// TEST/TestPackage/Templates/Internal/FB_BACnet_Server_NC01
// Notification Classes (Sample 01: Beckhoff)	
FUNCTION_BLOCK FB_BACnet_Server_NC01 EXTENDS FB_BACnet_View
VAR CONSTANT
	iAlarmModeFirst		: INT		:= 1;
	iAlarmModeLast		: INT		:= 3;
END_VAR
VAR
	// Event Typ "Alarm":
	aNCAlm_LifeSafety		: ARRAY[iAlarmModeFirst .. iAlarmModeLast] OF FB_BACnet_NC := [
								(
									iParent									:= THIS^,
									nObjectInstance							:= 12,
									nNotificationClass						:= 12,
									sObjectName								:= '\/NC12',
									sDescription							:= '\/Meldeklasse - Alarm Lebensgefahr (Einfach)',
									aAckRequired							:= [ TRUE, TRUE, FALSE ],
									aPriority								:= [ 10, 11, 12 ]),
								(
									iParent									:= THIS^,
									nObjectInstance							:= 11,
									nNotificationClass						:= 11,
									sObjectName								:= '\/NC11',
									sDescription							:= '\/Meldeklasse - Alarm Lebensgefahr (Standard)',
									aAckRequired							:= [ TRUE, TRUE, FALSE ],
									aPriority								:= [ 13, 14, 15 ]),
								(
									iParent									:= THIS^,
									nObjectInstance							:= 10,
									nNotificationClass						:= 10,
									sObjectName								:= '\/NC10',
									sDescription							:= '\/Meldeklasse - Alarm Lebensgefahr (Erweitert)',
									aAckRequired							:= [ TRUE, TRUE, TRUE ],
									aPriority								:= [ 16, 17, 18 ])
							];
							
	aNCAlm_Technical		: ARRAY[iAlarmModeFirst .. iAlarmModeLast] OF FB_BACnet_NC := [
								(
									iParent									:= THIS^,
									nObjectInstance							:= 22,
									nNotificationClass						:= 22,
									sObjectName								:= '\/NC22',
									sDescription							:= '\/Meldeklasse - Technischer Alarm (Einfach)',
									aAckRequired							:= [ TRUE, TRUE, FALSE ],
									aPriority								:= [ 20, 21, 22 ]),
								(
									iParent									:= THIS^,
									nObjectInstance							:= 21,
									nNotificationClass						:= 21,
									sObjectName								:= '\/NC21',
									sDescription							:= '\/Meldeklasse - Technischer Alarm (Standard)',
									aAckRequired							:= [ TRUE, TRUE, FALSE ],
									aPriority								:= [ 23, 24, 25 ]),
								(
									iParent									:= THIS^,
									nObjectInstance							:= 20,
									nNotificationClass						:= 20,
									sObjectName								:= '\/NC20',
									sDescription							:= '\/Meldeklasse - Technischer Alarm (Erweitert)',
									aAckRequired							:= [ TRUE, TRUE, TRUE ],
									aPriority								:= [ 26, 27, 28 ])
							];
							
	// Event Typ "Disturb":
	aNCDstb				: ARRAY[iAlarmModeFirst .. iAlarmModeLast] OF FB_BACnet_NC := [
								(
									iParent									:= THIS^,
									nObjectInstance							:= 52,
									nNotificationClass						:= 52,
									sObjectName								:= '\/NC52',
									sDescription							:= '\/Meldeklasse - Störung (Einfach)',
									aAckRequired							:= [ TRUE, TRUE, FALSE ],
									aPriority								:= [ 50, 51, 52 ]),
								(
									iParent									:= THIS^,
									nObjectInstance							:= 51,
									nNotificationClass						:= 51,
									sObjectName								:= '\/NC51',
									sDescription							:= '\/Meldeklasse - Störung (Standard)',
									aAckRequired							:= [ TRUE, TRUE, FALSE ],
									aPriority								:= [ 53, 54, 55 ]),
								(
									iParent									:= THIS^,
									nObjectInstance							:= 50,
									nNotificationClass						:= 50,
									sObjectName								:= '\/NC50',
									sDescription							:= '\/Meldeklasse - Störung (Erweitert)',
									aAckRequired							:= [ TRUE, TRUE, TRUE ],
									aPriority								:= [ 56, 57, 58 ])
							];
							
	// Event Typ "Maintenance":
	aNCMntn				: ARRAY[iAlarmModeFirst .. iAlarmModeLast] OF FB_BACnet_NC := [
								(
									iParent									:= THIS^,
									nObjectInstance							:= 92,
									nNotificationClass						:= 92,
									sObjectName								:= '\/NC92',
									sDescription							:= '\/Meldeklasse - Wartung (Einfach)',
									aAckRequired							:= [ TRUE, TRUE, FALSE ],
									aPriority								:= [ 90, 91, 92 ]),
								(
									iParent									:= THIS^,
									nObjectInstance							:= 91,
									nNotificationClass						:= 91,
									sObjectName								:= '\/NC91',
									sDescription							:= '\/Meldeklasse - Wartung (Standard)',
									aAckRequired							:= [ TRUE, TRUE, FALSE ],
									aPriority								:= [ 93, 94, 95 ]),
								(
									iParent									:= THIS^,
									nObjectInstance							:= 90,
									nNotificationClass						:= 90,
									sObjectName								:= '\/NC90',
									sDescription							:= '\/Meldeklasse - Wartung (Erweitert)',
									aAckRequired							:= [ TRUE, TRUE, TRUE ],
									aPriority								:= [ 96, 97, 98 ])
							];
							
	// Event Typ "Notification":
	aNCNtfy				: ARRAY[iAlarmModeFirst .. iAlarmModeLast] OF FB_BACnet_NC := [
								(
									iParent									:= THIS^,
									nObjectInstance							:= 132,
									nNotificationClass						:= 132,
									sObjectName								:= '\/NC132',
									sDescription							:= '\/Meldeklasse - Benachrichtigung (Einfach)',
									aAckRequired							:= [ TRUE, TRUE, FALSE ],
									aPriority								:= [ 130, 131, 132 ]),
								(
									iParent									:= THIS^,
									nObjectInstance							:= 131,
									nNotificationClass						:= 131,
									sObjectName								:= '\/NC131',
									sDescription							:= '\/Meldeklasse - Benachrichtigung (Standard)',
									aAckRequired							:= [ TRUE, TRUE, FALSE ],
									aPriority								:= [ 133, 134, 135 ]),
								(
									iParent									:= THIS^,
									nObjectInstance							:= 130,
									nNotificationClass						:= 130,
									sObjectName								:= '\/NC130',
									sDescription							:= '\/Meldeklasse - Benachrichtigung (Erweitert)',
									aAckRequired							:= [ TRUE, TRUE, TRUE ],
									aPriority								:= [ 136, 137, 138 ])
							];
							
	// Event Typ "Other":	
	aNCOthr				: ARRAY[iAlarmModeFirst .. iAlarmModeLast] OF FB_BACnet_NC := [
								(
									iParent									:= THIS^,
									nObjectInstance							:= 182,
									nNotificationClass						:= 182,
									sObjectName								:= '\/NC182',
									sDescription							:= '\/Meldeklasse - Sonstiges (Einfach)',
									aAckRequired							:= [ TRUE, TRUE, FALSE ],
									aPriority								:= [ 180, 181, 182 ]),
								(
									iParent									:= THIS^,
									nObjectInstance							:= 181,
									nNotificationClass						:= 181,
									sObjectName								:= '\/NC181',
									sDescription							:= '\/Meldeklasse - Sonstiges (Standard)',
									aAckRequired							:= [ TRUE, TRUE, FALSE ],
									aPriority								:= [ 183, 184, 185 ]),
								(
									iParent									:= THIS^,
									nObjectInstance							:= 180,
									nNotificationClass						:= 180,
									sObjectName								:= '\/NC180',
									sDescription							:= '\/Meldeklasse - Sonstiges (Erweitert)',
									aAckRequired							:= [ TRUE, TRUE, TRUE ],
									aPriority								:= [ 186, 187, 188 ])
							];
END_VAR
VAR
	iValTmp						: INT;
	iTemp						: INT;
END_VAR

SUPER^();

FOR iTemp := iAlarmModeFirst TO iAlarmModeLast DO
	aNCAlm_LifeSafety[iTemp]();
	aNCAlm_Technical[iTemp]();
	aNCDstb[iTemp]();
	aNCMntn[iTemp]();
	aNCNtfy[iTemp]();
	aNCOthr[iTemp]();
END_FOR

END_FUNCTION_BLOCK

// TEST/TestPackage/TestFBs/RT/FB_ArrayHtgCir
FUNCTION_BLOCK FB_ArrayHtgCir EXTENDS FB_BACnet_View
VAR_INPUT
	iCycleCount				: UINT;
END_VAR
VAR
	iTemp					: INT;
	aPlants					: ARRAY [1..MAX_PLANT] OF FB_Bnet_H_HtgCir_01;

	iCycleMOD				: UINT := 1;
	iLoopTo					: INT := MAX_PLANT;
END_VAR
VAR CONSTANT
	//MAX_PLANT				: INT := 29;			// Entspricht 1021 Ibjekte
	MAX_PLANT				: INT := 1;
END_VAR

SUPER^();

IF ((iCycleCount MOD iCycleMOD) = 0) THEN
	FOR iTemp := 1 TO iLoopTo DO
		aPlants[iTemp]();
	END_FOR
END_IF

METHOD FB_init : BOOL
VAR_INPUT
	bInitRetains : BOOL; // if TRUE, the retain variables are initialized (warm start / cold start)
	bInCopyCode : BOOL;  // if TRUE, the instance afterwards gets moved into the copy code (online change)
END_VAR
sObjectName		:= 'Test Heizkreise';
sDescription	:= 'Array mit vielen Heizkreisen';

FOR iTemp := 1 TO MAX_PLANT DO
	aPlants[iTemp].Parent		:= THIS^;
	aPlants[iTemp].sObjectName 	:= CONCAT('HtgCir', TO_STRING(iTemp));
	aPlants[iTemp].sDescription	:= CONCAT('Heizkreis ', TO_STRING(iTemp));
END_FOR
END_METHOD

END_FUNCTION_BLOCK

// TEST/TestPackage/TestFBs/RT/FB_ArrayTest
FUNCTION_BLOCK FB_ArrayTest EXTENDS FB_BACnet_View
VAR_INPUT
	iCycleCount				: UINT;
END_VAR
VAR					
	iTemp					: INT;
	BVObjects				: ARRAY [1..MAX_OBJECT] OF FB_BACnet_BV;

	iCycleMOD				: UINT := 1;
	iLoopTo					: INT := MAX_OBJECT;
END_VAR
VAR CONSTANT
	MAX_OBJECT : INT := 1000;
END_VAR

SUPER^();

IF ((iCycleCount MOD iCycleMOD) = 0) THEN
	FOR iTemp := 1 TO iLoopTo DO
		BVObjects[iTemp]();
	END_FOR
END_IF

METHOD FB_init : BOOL
VAR_INPUT
	bInitRetains : BOOL; // if TRUE, the retain variables are initialized (warm start / cold start)
	bInCopyCode : BOOL;  // if TRUE, the instance afterwards gets moved into the copy code (online change)
END_VAR
sObjectName		:= 'TestArray';
sDescription	:= 'Array mit vielen Objekten';

FOR iTemp := 1 TO MAX_OBJECT DO
	BVObjects[iTemp].Parent						:= THIS^;
//	BVObjects[iTemp].sObjectName 				:= CONCAT('BV üäß', TO_STRING(iTemp));
//	BVObjects[iTemp].sDescription				:= CONCAT('Binary Value üäß ', TO_STRING(iTemp));
//	
//	BVObjects[iTemp].sActiveText				:= '€ ÄÄÄ üß';
//	BVObjects[iTemp].sInactiveText				:= 'Money money $$ ÄÄÄ üß';
END_FOR
END_METHOD

END_FUNCTION_BLOCK

// TEST/TestPackage/TestFBs/FB_ClientTest
FUNCTION_BLOCK FB_ClientTest
VAR_INPUT CONSTANT
	AV_1 : FB_BACnetRM_AV := (Client:=Client,nObjectInstance:=1);
	AV_2 : FB_BACnetRM_AV := (Client:=Client,nObjectInstance:=2);
	AV_3 : FB_BACnetRM_AV := (Client:=Client,nObjectInstance:=3);
	AV_4 : FB_BACnetRM_AV := (Client:=Client,nObjectInstance:=4);
	AV_5 : FB_BACnetRM_AV := (Client:=Client,nObjectInstance:=5);
	AV_6 : FB_BACnetRM_AV := (Client:=Client,nObjectInstance:=6);
	AV_7 : FB_BACnetRM_AV := (Client:=Client,nObjectInstance:=7);
	AV_8 : FB_BACnetRM_AV := (Client:=Client,nObjectInstance:=8);
	AV_9 : FB_BACnetRM_AV := (Client:=Client,nObjectInstance:=9);
	AV_10: FB_BACnetRM_AV := (Client:=Client,nObjectInstance:=10);
	AV_11: FB_BACnetRM_AV := (Client:=Client,nObjectInstance:=11);
	AV_12: FB_BACnetRM_AV := (Client:=Client,nObjectInstance:=12);
END_VAR
VAR
	Client : FB_BACnet_Client := (eReadMode:=E_BACnet_CommMode.eRp);
END_VAR

Client();
AV_1();
AV_2();
AV_3();
AV_4();
AV_5();
AV_6();
AV_7();
AV_8();
AV_9();
AV_10();
AV_11();
AV_12();

END_FUNCTION_BLOCK

// TEST/TestPackage/_MAIN
PROGRAM _MAIN
VAR
	wDummy			AT %I*	: WORD;
	
	bKillMe11				: BOOL;
END_VAR
VAR
	bInit					: BOOL := TRUE;
	nCycles					: UDINT;
END_VAR
VAR
	bManualWritePersistent	: BOOL;
	tAutoWritePersistent	: TON						:= (PT := T#20S);
	wPersistentData			: FB_WritePersistentData	:= (PORT:=TwinCAT_SystemInfoVarList._AppInfo.AdsPort, TMOUT:=T#1S, MODE:=E_PersistentMode.SPDM_2PASS);
END_VAR

nCycles := (nCycles+1);
IF (bInit) THEN
	bInit := FALSE;
END_IF

// Persistent data:
tAutoWritePersistent(IN := (NOT tAutoWritePersistent.Q));
IF (bManualWritePersistent) OR (tAutoWritePersistent.Q) THEN
	bManualWritePersistent := FALSE;
	wPersistentData(START:=TRUE);
ELSE
	wPersistentData();
	IF (NOT wPersistentData.BUSY) THEN
		wPersistentData.START:=FALSE;
	END_IF
END_IF



// Sample programs:
// Uncomment to execute samples:
//////////////////////////////////////////////////

//CLIENT();
//PLANT_DEMO();
//MAIN_PRG02();
//PERFORMANCE();
//PERFORMANCE_MIX();
RT();
//DYN_OBJECTS();

END_PROGRAM

// TEST/TestPackage/PLANT_DEMO
PROGRAM PLANT_DEMO
VAR
	fbStatHeatingCir	: FB_Bnet_H_HtgCir_01		:= (sObjectName				:= 'HTGCIR01',
														sDescription			:= '\/Statische Heizung',
														Pu := (
															sObjectName			:= '\/TEST01_PU01',
															Dst := (
																sObjectName		:= '\/DST01')));
																
	fbFlHeatingCir		: FB_Bnet_H_HtgCir_01		:= (sObjectName				:= 'HTGCIR02',
														sDescription			:= '\/Fußbodenheizung');
																
	fbRoom3				: FB_Bnet_H_HtgCir_01		:= (sObjectName				:= 'HTGCIR03',
														sDescription			:= '\/Heizung Raum 3');
END_VAR

fbStatHeatingCir();
fbFlHeatingCir();
fbRoom3();

METHOD FB_init : BOOL
VAR_INPUT
	bInitRetains : BOOL; // if TRUE, the retain variables are initialized (warm start / cold start)
	bInCopyCode : BOOL;  // if TRUE, the instance afterwards gets moved into the copy code (online change)
END_VAR
fbStatHeatingCir.Pu.sObjectName			:= '\/TEST01_PU01';
fbStatHeatingCir.Pu.sObjectName			:= '\/TEST01_PU01';
fbStatHeatingCir.Pu.sObjectName			:= '\/TEST01_PU01';
fbStatHeatingCir.Pu.sObjectName			:= '\/TEST01_PU01';
fbStatHeatingCir.Pu.sObjectName			:= '\/TEST01_PU01';
END_METHOD

END_PROGRAM

// TEST/TestPackage/PERFORMANCE
PROGRAM PERFORMANCE
// Test für RT-Objekte:
VAR
	//fbHtgCirArray : FB_ArrayHtgCir;
	fbObjArray : FB_ArrayTest;
	
	bStop : BOOL;
END_VAR


// Test für RT-Objekte:
//fbHtgCirArray();
IF NOT bStop THEN
	fbObjArray();
END_IF

END_PROGRAM

// TEST/TestPackage/RT
// Dieses Programm testet die RT-Bausteine, welche der LIB-Variante nachempfunden sind.
PROGRAM RT
VAR
	bKillMe1 : BOOL;
	_hRes : HRESULT;
	tTemp : T_MaxString;
END_VAR
VAR_INPUT
	nLibNode_UpdateCount				: UDINT;
	fbLibNode							: FB_BACnet_View := (
											eNodeType								:= E_BACnet_NodeType.eArea,
											sObjectName								:= '\/LibNde',
											sDescription							:= '\/Test RT-Lib Node');
END_VAR
// --- Analog: ---------------------------------------------------------------------------------------------------------------------------------------
VAR_INPUT
	fbANode								: FB_BACnet_View := (
											iParent									:= fbLibNode,
											eNodeType								:= E_BACnet_NodeType.eArea,
											sObjectName								:= '\/A',
											sDescription							:= '\/Analog');

	AV									: FB_BACnet_AV := (
											iParent									:= fbANode,
											nObjectInstance							:= 115,
											sObjectName								:= '\/AV 01',
											sDescription							:= '\/Analog Value Test 1 öäü',
											eUnit									:= E_BA_Unit.eOther_Percent,
											bHighLimitEnable						:= TRUE,
											fHighLimit								:= 50,
											bLowLimitEnable							:= TRUE,
											fLowLimit								:= 10,
											nNotificationClass						:= 11,
											aEventEnable							:= [ TRUE, TRUE, FALSE ],
											aEventMessageTextsConfig				:= [ '\/Ausgelöst', '\/Fehler', '\/Normal' ]);

	// Intention:						Value
	// Priorities						5P
	AV5P_TestEnSfty				AT %I*	: BOOL; // Test: Safety ist von PLC aus immer beschaltet
	AV5P								: FB_BACnet_AV_5P := (
											iParent									:= fbANode,
											sDescription							:= '\/Analog Value 5Prio',
											eUnit									:= E_BA_Unit.eOther_Percent,
											bEnPgm									:= TRUE,
											fValPgm									:= 10.0);
											
	// Intention:						Value for Display
	// Operation:						Display
	AVDsp								: FB_BACnet_AV_Disp := (
											iParent									:= fbANode,
											sDescription							:= '\/Test AV Display',
											eUnit									:= E_BA_Unit.eOther_Percent);	
	
	// Intention:						Value for Setpoint
	// Operation:						Setpoint
	AVSp								: FB_BACnet_AV_Setp := (
											iParent									:= fbANode,
											sDescription							:= '\/Test AV Setpoint',
											eUnit									:= E_BA_Unit.eTime_Hours,
											fValue									:= 168);

	AI_TSenRaw_State			AT %I*	: USINT;
	AI_TSenRaw_DataIn			AT %I*	: INT;
	AI_TSenRaw							: FB_BACnet_AI_Raw := (
											iParent									:= fbANode,
											sDescription							:= '\/Test AI Fühler (Raw)',
											sDeviceType								:= 'Fühler',
											eUnit									:= E_BA_Unit.eOther_Percent,
											fResolution								:= 0.003814755,
											fScaleOffset							:= 0.0,
											fHighLimit								:= 150,
											fLowLimit								:= -500,
											nNotificationClass						:= 10,
											aEventEnable							:= [ TRUE, TRUE, FALSE ],
											aEventMessageTextsConfig				:= [ '\/Ausgelöst', '\/Fehler', '\/Normal' ]);

	// Intention:						Input
	// Hardware:						Process
	AI_TSenProc_Value					: REAL := 50.0;
	AI_TSenProc							: FB_BACnet_AI := (
											iParent									:= fbANode,
											sDescription							:= '\/Test AI (Prozesswert)',
											eUnit									:= E_BA_Unit.eOther_Percent,
											fHighLimit								:= 150,
											fLowLimit								:= -500,
											nNotificationClass						:= 10,
											aEventEnable							:= [ TRUE, TRUE, FALSE ],
											aEventMessageTextsConfig				:= [ '\/Ausgelöst', '\/Fehler', '\/Normal' ]);

	// Intention:						Input
	// Hardware:						I/O
	AI_TSenIO_IOBusState		AT %Q*	: UINT := 0;
	AI_TSenIO							: FB_BACnet_AI_IO := (
											iParent									:= fbANode,
											sDescription							:= '\/Test AI Fühler (IO)',
											sDeviceType								:= 'Fühler',
											eUnit									:= E_BA_Unit.eOther_Percent,
											fResolution								:= 0.003814755,
											fScaleOffset							:= 0.0,
											fHighLimit								:= 150,
											fLowLimit								:= -500,
											nIoBusNr								:= 0,
											nNotificationClass						:= 10,
											aEventEnable							:= [ TRUE, TRUE, FALSE ],
											aEventMessageTextsConfig				:= [ '\/Ausgelöst', '\/Fehler', '\/Normal' ]);

	// Intention:						Input for Display
	// Operation:						Display
	// Hardware:						I/O
	// Parameter:						EventDetectionEnable = FALSE
	AIDsp_TSenIO						: FB_BACnet_AI_IO := (
											iParent									:= fbANode,
											sDescription							:= '\/Test AI Display Fühler (IO)',
											sDeviceType								:= 'Fühler',
											eUnit									:= E_BA_Unit.eOther_Percent,
											bEventDetectionEnable					:= FALSE);

	AO_Cmd_RlbtyPgm						: E_BA_Reliability;
	AO_Cmd_RawOvrrd						: BOOL;
	AO_Cmd								: FB_BACnet_AO := (
											iParent									:= fbANode,
											sDescription							:= '\/Befehl AO',
											sDeviceType								:= 'Ausgang',
											eUnit									:= E_BA_Unit.eOther_Percent,
											fResolution								:= 0.003051851,
											fScaleOffset							:= 0.0,
											fHighLimit								:= 150,
											fLowLimit								:= -50,
											nNotificationClass						:= 10,
											aEventEnable							:= [ TRUE, TRUE, FALSE ],
											aEventMessageTextsConfig				:= [ '\/Ausgelöst', '\/Fehler', '\/Normal' ]);

	AO_CmdRaw_Out				AT %Q*	: INT;
	AO_CmdRaw							: FB_BACnet_AO_Raw := (
											iParent									:= fbANode,
											sDescription							:= '\/Befehl AO (Raw)',
											sDeviceType								:= 'Ausgang',
											eUnit									:= E_BA_Unit.eOther_Percent,
											fResolution								:= 0.003051851,
											fScaleOffset							:= 0.0,
											fHighLimit								:= 150,
											fLowLimit								:= -50,
											nNotificationClass						:= 10,
											aEventEnable							:= [ TRUE, TRUE, FALSE ],
											aEventMessageTextsConfig				:= [ '\/Ausgelöst', '\/Fehler', '\/Normal' ]);

	AO_CmdIORaw							: FB_BACnet_AO_IO := (
											iParent									:= fbANode,
											sDescription							:= '\/Befehl AO (IO)',
											sDeviceType								:= 'Ausgang',
											eUnit									:= E_BA_Unit.eOther_Percent,
											fResolution								:= 0.003051851,
											fScaleOffset							:= 0.0,
											fHighLimit								:= 150,
											fLowLimit								:= -50,
											nNotificationClass						:= 10,
											aEventEnable							:= [ TRUE, TRUE, FALSE ],
											aEventMessageTextsConfig				:= [ '\/Ausgelöst', '\/Fehler', '\/Normal' ]);

	AO_Cmd5P_RlbtyPgm					: E_BA_Reliability;
	AO_Cmd5P_RawOvrrd					: BOOL;
	AO_Cmd5P							: FB_BACnet_AO_5P := (
											iParent									:= fbANode,
											sDescription							:= '\/Analog Befehl 5Prio',
											eUnit									:= E_BA_Unit.eOther_Percent);

	AO_CmdRaw5P_State			AT %I*	: USINT;
	AO_CmdRaw5P_Out				AT %Q*	: INT;
	AO_CmdRaw5P							: FB_BACnet_AO_Raw5P := (
											iParent									:= fbANode,
											sDescription							:= '\/Analog Befehl 5Prio (Raw)',
											eUnit									:= E_BA_Unit.eOther_Percent);

	// Intention:						Output
	// Hardware:						I/O
	// Priorities						5P
	AO_CmdIO5P							: FB_BACnet_AO_IO5P := (
											iParent									:= fbANode,
											sDescription							:= '\/Analog Befehl 5Prio (IO)',
											eUnit									:= E_BA_Unit.eOther_Percent);

	// Intention:						Output for Display
	// Operation:						Display
	// Hardware:						I/O
	// Parameter:						EventDetectionEnable = FALSE
	AODisp_CmdIO5P						: FB_BACnet_AO_IO5P := (
											iParent									:= fbANode,
											sDescription							:= '\/Analog Befehl 5Prio Display (IO)',
											eUnit									:= E_BA_Unit.eOther_Percent,
											bEventDetectionEnable					:= FALSE);
											
	AO_CmdIO							: FB_BACnet_AO_IO := (
											iParent									:= fbANode,
											sDescription							:= '\/Analog Befehl (IO)',
											eUnit									:= E_BA_Unit.eOther_Percent);
END_VAR
// --- Binary: ---------------------------------------------------------------------------------------------------------------------------------------
VAR_INPUT
	fbBNode								: FB_BACnet_View := (
											iParent									:= fbLibNode,
											eNodeType								:= E_BACnet_NodeType.eArea,
											sObjectName								:= '\/B',
											sDescription							:= '\/Binary');
											
	BV									: FB_BACnet_BV := (
											iParent									:= fbBNode,
											nObjectInstance							:= 99,
											sDescription							:= '\/Test BV',
											bAlarmValue								:= FALSE);

	// Intention:						Value
	// Priorities						5P
	BV5P								: FB_BACnet_BV_5P := (
											iParent									:= fbBNode,
											sDescription							:= '\/Binary Value 5Prio');
											
	// Intention:						Value for Display
	// Operation:						Display
	BVDsp								: FB_BACnet_BV_Disp := (
											iParent									:= fbBNode,
											sDescription							:= '\/Test BV Display',
											sInactiveText							:= 'Aus',
											sActiveText								:= 'Ein');
	
	// Intention:						Value for Setpoint
	// Operation:						Setpoint
	BVSp								: FB_BACnet_BV_Setp := (
											iParent									:= fbBNode,
											sDescription							:= '\/Test BV Setpoint',
											sInactiveText							:= 'Aus',
											sActiveText								:= 'Ein',
											bValue									:= TRUE);

	BI_DstbRaw_In				AT %I*	: BOOL;
	BI_DstbRaw							: FB_BACnet_BI_Raw := (
											iParent									:= fbBNode,
											sDescription							:= '\/Test BI Disturb (Raw)',
											sDeviceType								:= 'Sicherung',
											sInactiveText							:= 'Normal',
											sActiveText								:= 'Ausgelöst',
											ePolarity								:= E_BA_Polarity.eReverse,
											nNotificationClass						:= 10,
											aEventEnable							:= [ TRUE, TRUE, FALSE ],
											aEventMessageTextsConfig				:= [ '\/Ausgelöst', '\/Fehler', '\/Normal' ]);
											
	// Intention:						Input
	// Hardware:						I/O
	BI_DstbIO							: FB_BACnet_BI_IO := (
											iParent									:= fbBNode,
											sDescription							:= '\/Test BI Disturb (IO)',
											sDeviceType								:= 'Sicherung',
											sInactiveText							:= 'Normal',
											sActiveText								:= 'Ausgelöst',
											ePolarity								:= E_BA_Polarity.eReverse,
											nNotificationClass						:= 10,
											aEventEnable							:= [ TRUE, TRUE, FALSE ],
											aEventMessageTextsConfig				:= [ '\/Ausgelöst', '\/Fehler', '\/Normal' ]);

	// Intention:						Input for Display
	// Operation:						Display
	// Hardware:						I/O
	// Parameter:						EventDetectionEnable = FALSE
	BIDsp_SwiIO							: FB_BACnet_BI_IO := (
											iParent									:= fbBNode,
											sDescription							:= '\/Test BI Schalter Display (IO)',
											sDeviceType								:= 'Sicherung',
											sInactiveText							:= 'Normal',
											sActiveText								:= 'Ausgelöst',
											ePolarity								:= E_BA_Polarity.eReverse,
											bEventDetectionEnable					:= FALSE);

	BO_Cmd_RlbtyPgm						: E_BA_Reliability;
	BO_Cmd_RawOvrrd						: BOOL;
	BO_Cmd								: FB_BACnet_BO := (
											iParent									:= fbBNode,
											sDescription							:= '\/Test BO Befehl',
											sInactiveText							:= 'Aus',
											sActiveText								:= 'Ein');
											
	BO_CmdRaw_Out				AT %Q*	: BOOL;
	BO_CmdRaw							: FB_BACnet_BO_Raw := (
											iParent									:= fbBNode,
											sDescription							:= '\/Test BO Befehl (Raw)',
											sInactiveText							:= 'Aus',
											sActiveText								:= 'Ein');
											
	BO_CmdIO							: FB_BACnet_BO_IO := (
											iParent									:= fbBNode,
											sDescription							:= '\/Test BO Befehl (IO)',
											sInactiveText							:= 'Aus',
											sActiveText								:= 'Ein');

	BO_Cmd5P_RlbtyPgm					: E_BA_Reliability;
	BO_Cmd5P_RawOvrrd					: BOOL;
	BO_Cmd5P							: FB_BACnet_BO_5P := (
											iParent									:= fbBNode,
											sDescription							:= '\/Test BO Befehl 5Prio',
											sInactiveText							:= 'Aus',
											sActiveText								:= 'Ein',
											nTimeDelay								:= 3,
											nNotificationClass						:= 10,
											aEventEnable							:= [ TRUE, TRUE, FALSE ],
											aEventMessageTextsConfig				:= [ '\/Ausgelöst', '\/Fehler', '\/Normal' ]);
											
	BO_CmdRaw5P_Feedback		AT %I*	: BOOL;
	BO_CmdRaw5P_OverrIO			AT %I*	: BOOL;
	BO_CmdRaw5P_Out				AT %Q*	: BOOL;
	BO_CmdRaw5P							: FB_BACnet_BO_Raw5P := (
											iParent									:= fbBNode,
											sDescription							:= '\/Test BO Befehl 5Prio (Raw)',
											sInactiveText							:= 'Aus',
											sActiveText								:= 'Ein',
											nTimeDelay								:= 3,
											nNotificationClass						:= 10,
											aEventEnable							:= [ TRUE, TRUE, FALSE ],
											aEventMessageTextsConfig				:= [ '\/Ausgelöst', '\/Fehler', '\/Normal' ]);
											
	// Intention:						Output
	// Hardware:						I/O
	// Priorities						5P
	BO_CmdIO5P							: FB_BACnet_BO_IO5P := (
											iParent									:= fbBNode,
											sDescription							:= '\/Test BO Befehl 5Prio (IO)',
											sInactiveText							:= 'Aus',
											sActiveText								:= 'Ein',
											nTimeDelay								:= 3,
											nNotificationClass						:= 10,
											aEventEnable							:= [ TRUE, TRUE, FALSE ],
											aEventMessageTextsConfig				:= [ '\/Ausgelöst', '\/Fehler', '\/Normal' ]);
											
	// Intention:						Output for Display
	// Operation:						Display
	// Hardware:						I/O
	// Parameter:						EventDetectionEnable = FALSE
	BODisp_CmdIO5P						: FB_BACnet_BO_IO5P := (
											iParent									:= fbBNode,
											sDescription							:= '\/Test BO Befehl 5Prio Display (IO)',
											sInactiveText							:= 'Aus',
											sActiveText								:= 'Ein',
											bEventDetectionEnable					:= FALSE);
END_VAR
// --- Multistate: ---------------------------------------------------------------------------------------------------------------------------------------
VAR_INPUT
	fbMNode								: FB_BACnet_View := (
											iParent									:= fbLibNode,
											eNodeType								:= E_BACnet_NodeType.eArea,
											sObjectName								:= '\/M',
											sDescription							:= '\/Multistate');
											
	MV									: FB_BACnet_MV := (
											iParent									:= fbMNode,
											nObjectInstance							:= 99,
											sDescription							:= '\/Test MV',
											aAlarmValues							:= [ 1, 2 ],
											aFaultValues							:= [ 3 ],
										//	sStateText								:= [ 'Aus', 'Stufe 1', 'Stufe 2']);
										//	sStateText								:= [ 'Aus', 'Stufe 1', 'Stufe 2', 'Stufe 3', 'Stufe 4', 'Stufe 5', 'Stufe 6', 'Stufe 7', 'Stufe 8', 'Stufe 9', 'Stufe 10', 'Stufe 11', 'Stufe 12', 'Stufe 13', 'Stufe 14', 'Stufe 15' ]);
											sStateText								:= [ 'Aus', 'Stufe 1', 'Stufe 2', 'Stufe 3', 'Stufe 4', 'Stufe 5', 'Stufe 6', 'Stufe 7', 'Stufe 8', 'Stufe 9', 'Stufe 10' ]);

	// Intention:						Value
	// Priorities						5P
	MV5P								: FB_BACnet_MV_5P := (
											iParent									:= fbMNode,
											sDescription							:= '\/Test MV 5Prio',
											sStateText								:= [ 'Aus', 'Stufe 1', 'Stufe 2' ]);

	// Intention:						Value for Display
	// Operation:						Display
	MVDsp								: FB_BACnet_MV_Disp := (
											iParent									:= fbMNode,
											sDescription							:= '\/Test MV Display',
											sStateText								:= [ 'Wert 11', 'Wert 22' ]);
	
	// Intention:						Value for Setpoint
	// Operation:						Setpoint
	MVSp								: FB_BACnet_MV_Setp := (
											iParent									:= fbMNode,
											sDescription							:= '\/Test MV Display',
											sStateText								:= [ 'Auto', 'Aus', 'Ein' ],
											nValue									:= 2);

	MI_StateRaw_In						: UDINT;
	MI_StateRaw							: FB_BACnet_MI_Raw := (
											iParent									:= fbMNode,
											sDescription							:= '\/Test MI State (Raw)',
											sDeviceType								:= 'Gerät',
											aStateText								:= [ 'Störung 1', 'Störung 2', 'Fehler', 'Normal' ],
											aAlarmValues							:= [ 1, 2 ],
											aFaultValues							:= [ 3 ],
											nNotificationClass						:= 10,
											aEventEnable							:= [ TRUE, TRUE, FALSE ],
											aEventMessageTextsConfig				:= [ '\/Ausgelöst', '\/Fehler', '\/Normal' ]);

	// Intention:						Input
	// Hardware:						I/O
	MI_StateIO							: FB_BACnet_MI_IO := (
											iParent									:= fbMNode,
											sDescription							:= '\/Test MI State (IO)',
											sDeviceType								:= 'Gerät',
											aStateText								:= [ 'Aus', 'Stufe 1', 'Stufe 2', 'Stufe 3', 'Stufe 4' ],
											aAlarmValues							:= [ 3, 4 ],
											aFaultValues							:= [ 5 ],
											nNotificationClass						:= 10,
											aEventMessageTextsConfig				:= [ '\/Ausgelöst', '\/Fehler', '\/Normal' ]
										);
										
	// Intention:						Input for Display
	// Operation:						Display
	// Hardware:						I/O
	// Parameter:						EventDetectionEnable = FALSE
	MIDsp_Swi_StateRaw_In				: UDINT;
	MIDsp_Swi_StateRaw					: FB_BACnet_MI_Raw := (
											iParent									:= fbMNode,
											sDescription							:= '\/Test MI State (Raw)',
											sDeviceType								:= 'Gerät',
											aStateText								:= [ 'Störung 1', 'Störung 2', 'Fehler', 'Normal' ],
											bEventDetectionEnable					:= FALSE);

	MO_Cmd_RawOvrrd						: BOOL;
	MO_Cmd								: FB_BACnet_MO := (
											iParent									:= fbMNode,
											sDescription							:= '\/Test MO Befehl',
											sStateText								:= [ 'Stufe 1', 'Stufe 2', 'Aus' ]);

	MO_CmdRaw_Out						: UDINT;
	MO_CmdRaw							: FB_BACnet_MO_Raw := (
											iParent									:= fbMNode,
											sDescription							:= '\/Test MO Befehl (Raw)',
											sStateText								:= [ 'Stufe 1', 'Stufe 2', 'Aus' ]);

	MO_5P_RawOvrrd						: BOOL;
	MO_5P								: FB_BACnet_MO_5P := (
											iParent									:= fbMNode,
											sDescription							:= '\/Test MO Befehl 5Prio (Raw)',
											sStateText								:= [ 'Stufe 1', 'Stufe 2', 'Aus' ]);

	// Intention:						Output
	// Hardware:						I/O
	// Priorities						5P
	MO_Raw5P_Out						: UDINT;
	MO_Raw5P							: FB_BACnet_MO_Raw5P := (
											iParent									:= fbMNode,
											sDescription							:= '\/Test MO Befehl 5Prio (Raw)',
											sStateText								:= [ 'Stufe 1', 'Stufe 2', 'Aus' ]);

	MODisp_Raw5P_Out					: UDINT;
	MODisp_Raw5P						: FB_BACnet_MO_Raw5P := (
											iParent									:= fbMNode,
											sDescription							:= '\/Test MO Befehl 5Prio (Raw)',
											sStateText								:= [ 'Stufe 1', 'Stufe 2', 'Aus' ],
											bEventDetectionEnable					:= FALSE);
											

	// Intention:						Output for Display
	// Operation:						Display
	// Hardware:						I/O
	// Parameter:						EventDetectionEnable = FALSE
	MODisp_IO5P							: FB_BACnet_MO_IO5P := (
											iParent									:= fbMNode,
											sDescription							:= '\/Test MO Befehl (IO)',
											sStateText								:= [ 'Aus', 'Stufe 1', 'Stufe 2', 'Stufe 3', 'Stufe 4' ],
											bEventDetectionEnable					:= FALSE
										);
END_VAR
// --- Misc: ---------------------------------------------------------------------------------------------------------------------------------------
VAR_INPUT		
	fbMscNode							: FB_BACnet_View := (
											iParent									:= fbLibNode,
											eNodeType								:= E_BACnet_NodeType.eArea,
											sObjectName								:= '\/Misc',
											sDescription							:= '\/Miscellaneous');
											
	File01								: FB_BACnet_File := (
											iParent									:= fbMscNode,
											sDescription							:= '\/My File');
											
	Dev01								: FB_BACnet_Device := (
											iParent									:= fbMscNode,
											sDescription							:= '\/My Device',
											sLocation								:= 'Verl');
											
	Loop								: FB_BACnet_Loop := (
											iParent									:= fbMscNode,
											sDescription							:= '\/Test Loop',
											eOutputUnit								:= E_BA_Unit.eOther_Percent,
											eAction									:= E_BA_Action.eReverse,
											fProportionalConstant					:= 5.0,
											fIntegralConstant						:= 180,
											nNotificationClass						:= 10,
											aEventEnable							:= [ FALSE, FALSE, FALSE ],
											aEventMessageTextsConfig				:= [ '\/Überschritten', '\/Fehler', '\/Normal' ]);

	fbLoopRefNode						: FB_BACnet_View := (
											iParent									:= fbMscNode,
											sObjectName								:= '\/LoopRef',
											sDescription							:= '\/Loop Reference');
	LoopRef_Setpt						: FB_BACnet_AV_Setp := (
											iParent									:= fbLoopRefNode,
											fValue									:= 20);
	LoopRef_CtrlVar						: FB_BACnet_AV_Setp := (
											iParent									:= fbLoopRefNode,
											fValue									:= 18);
	LoopRef_Y							: FB_BACnet_AV_Disp := (
											iParent									:= fbLoopRefNode);
	LoopRef								: FB_BACnet_Loop_Ref := (
											iParent									:= fbLoopRefNode,
											sDescription							:= '\/Test Loop Reference',
											stControlledVariableReference			:= F_BACnet_Reference(LoopRef_CtrlVar, PropPresentValue),
											stSetpointReference						:= F_BACnet_Reference(LoopRef_Setpt, PropPresentValue),
											stManipulatedVariableReference			:= F_BACnet_Reference(LoopRef_Y, PropPresentValue),
											eOutputUnit								:= E_BA_Unit.eOther_Percent,
											eAction									:= E_BA_Action.eReverse,
											fProportionalConstant					:= 5.0,
											fIntegralConstant						:= 180,
											fDeadband								:= 99.0,
											fErrorLimit								:= 99.0,
											nNotificationClass						:= 10,
											aEventEnable							:= [ FALSE, FALSE, FALSE ],
											aEventMessageTextsConfig				:= [ '\/Überschritten', '\/Fehler', '\/Normal' ]);

	CAL01								: FB_BACnet_Cal := (
											iParent									:= fbMscNode,
											sDescription							:= '\/Kalender 1',
											aDateList := [(
												eType								:= E_BA_DateValChoice.eDate,
												uDate								:= F_BA_DateVal(2020,E_BA_Month.eApril,10)),
											(
												eType								:= E_BA_DateValChoice.eDateRange,
												uDate								:= F_BA_DateRangeVal(nFromYear:=2020,E_BA_Month.eApril,10, nToYear:=2021,E_BA_Month.eMay,11)),
											(
												eType								:= E_BA_DateValChoice.eWeekNDay,
												uDate								:= F_BA_WeekNDayVal(E_BA_Weekday.eFriday, E_BA_Week.eWeek1, E_BA_Month.eFebruary))
											]);
	CAL02								: FB_BACnet_Cal := (
											iParent									:= fbMscNode,
											sDescription							:= '\/Kalender 2');
	CAL03								: FB_BACnet_Cal := (
											iParent									:= fbMscNode,
											sDescription							:= '\/Kalender 3');
	
	// Intention:						Scheduler for analog values
	// Parameter:						tWeek = F_BACnet_SchedWeeklyXxA(...)
	//									tCalendar = [(...), (...), (...)]
	//									tException = [(..., F_BACnet_SchedEntryXxA(...)), (..., F_BACnet_SchedEntryXxA(...)), (..., F_BACnet_SchedEntryXxA(...)), (..., [10:00h > 1.0],[11:00h > null])]
	SchedA								: FB_BACnet_SchedA := (
											iParent									:= fbMscNode,
											sDescription							:= '\/Scheduler Analog',
											aObjectPropertyReferences := [
												(iObject := AVSp, ePropertyId := PropPresentValue)
											],
											aWeek									:= F_BACnet_SchedWeekly3xA(E_BA_Weekday.eMonday, E_BA_Weekday.eFriday, T#0H, 0.0, T#6H, 5.0, T#20H, 0.0),
											aCalendar := [(
												iRefCalendar						:= CAL01,
												aEntry								:= F_BACnet_SchedEntry1xA(T#0H, 2.0)),
											(
												iRefCalendar						:= CAL02,
												aEntry								:= F_BACnet_SchedEntry1xA(T#10H, 3.4)),
											(
												iRefCalendar						:= CAL03,
												aEntry								:= F_BACnet_SchedEntry3xA(T#0H, 5, T#6H, 7, T#20H, 8))
											],
											aException := [(
												eType								:= E_BA_DateValChoice.eDate,
												uDate								:= F_BA_DateVal(2020,E_BA_Month.eApril,10),
												aEntry								:= F_BACnet_SchedEntry1xA(T#0H, 0.0)),
											(
												eType								:= E_BA_DateValChoice.eDateRange,
												uDate								:= F_BA_DateRangeVal(nFromYear:=2020,E_BA_Month.eApril,10, nToYear:=2021,E_BA_Month.eMay,11),
												aEntry								:= F_BACnet_SchedEntry3xA(T#0H, 0.0, T#6H, 5.0, T#20H, 0.0)),
											(
												eType								:= E_BA_DateValChoice.eWeekNDay,
												uDate								:= F_BA_WeekNDayVal(E_BA_Weekday.eFriday, E_BA_Week.eWeek1, E_BA_Month.eFebruary),
												aEntry								:= F_BACnet_SchedEntry3xA(T#0H, 0.0, T#6H, 5.0, T#20H, 0.0)),
											(
												eType								:= E_BA_DateValChoice.eDate,
												uDate								:= F_BA_DateVal(2019,E_BA_Month.eJune,20),
												aEntry := [(
													eState							:= E_BA_SchedEntryState.eValue,
													stTime							:= F_BA_ToSTTime(T#10H),
													uValue							:= F_BA_RVal(1.0)),
												(
													eState							:= E_BA_SchedEntryState.eNull,
													stTime							:= F_BA_ToSTTime(T#11H)
												)]
											)]);
	
	// Intention:						Scheduler for boolean values
	// Parameter:						tWeek = F_BACnet_SchedWeeklyXxB(...)
	//									tCalendar = F_BACnet_SchedCalendar(...)
	SchedB_AssignTestCal2Reference		: BOOL;
	SchedB								: FB_BACnet_SchedB := (
											iParent									:= fbMscNode,
											sDescription							:= '\/Scheduler Bool',
											aWeek									:= F_BACnet_SchedWeekly3xB(E_BA_Weekday.eMonday, E_BA_Weekday.eFriday, T#0H, FALSE, T#6H, TRUE, T#20H, FALSE),
											aCalendar := [(
												iRefCalendar						:= CAL01,
												aEntry								:= F_BACnet_SchedEntry1xB(T#0H, FALSE)
											),(
												iRefCalendar						:= CAL02,
												aEntry								:= F_BACnet_SchedEntry1xB(T#10H, TRUE)
											),(
												iRefCalendar						:= CAL03,
												aEntry								:= F_BACnet_SchedEntry3xB(T#0H, FALSE, T#6H, TRUE, T#20H, FALSE)
											)]);
	
	// Intention:						Scheduler for multistate values
	SchedM								: FB_BACnet_SchedM := (
											iParent									:= fbMscNode,
											sDescription							:= '\/Scheduler Multistate',
											aWeek									:= F_BACnet_SchedWeekly3xM(E_BA_Weekday.eMonday, E_BA_Weekday.eFriday, T#0H, 1, T#6H, 2, T#20H, 1));
	
	EventLog_NC11						: FB_BACnet_ELog := (
											iParent									:= fbMscNode,
											sDescription							:= '\/Event Log für NC11',
											nObjectInstance							:= 11,
											bLogEnable								:= TRUE,
											aEventEnable							:= [ TRUE, TRUE, FALSE ],
											aEventMessageTextsConfig				:= [ '\/Überschritten', '\/Fehler', '\/Normal' ]);
	EventLog_NC12						: FB_BACnet_ELog := (
											iParent									:= fbMscNode,
											sDescription							:= '\/Event Log für NC12',
											nObjectInstance							:= 12,
											bLogEnable								:= TRUE,
											aEventEnable							:= [ TRUE, TRUE, FALSE ],
											aEventMessageTextsConfig				:= [ '\/Überschritten', '\/Fehler', '\/Normal' ]);

	// (BETA) ... TODO
	// SCHED_Multistate : FB_BACnet_SchedMultistate;
	
	TLog_AssignTestReference			: BOOL;
	TLog_ReadReference					: BOOL;
	TLog_LogReferenceInfo				: BOOL;
	TLog								: FB_BACnet_TLog := (
											iParent									:= fbMscNode,
											sDescription							:= '\/Trend',
											nNotificationClass						:= 11,
											aEventEnable							:= [ TRUE, TRUE, FALSE ],
											aEventMessageTextsConfig				:= [ '\/Überschritten', '\/Fehler', '\/Normal' ],
											stStartTime								:= F_BA_ToSTDateTime(DT#2010-01-01-00:00),
											bLogEnable								:= TRUE,
											stObjectPropertyReference				:= F_BACnet_Reference(AVSp, PropPresentValue));
											
	TLogCov								: FB_BACnet_TLog := (
											iParent									:= fbMscNode,
											sDescription							:= '\/Trend Cov',
											bLogEnable								:= TRUE,
											stObjectPropertyReference				:= F_BACnet_Reference(AVSp, PropPresentValue),			
											eLoggingType 							:= E_BA_LoggingType.eCOV, 							
											nCOVResubscriptionInterval				:= 600,
											stClientCOV := (
												eChoice								:= E_BACnet_ClientCOVChoice.eCovReal,
												fIncrement							:= 1.0
											));
											
	TLogNoRef							: FB_BACnet_TLog := (
											iParent									:= fbMscNode,
											sDescription							:= '\/Trend (Ohne Referenz)');
	TLogM								: FB_BACnet_TLM := (
											iParent									:= fbMscNode,
											sDescription							:= '\/Trend Multiple',
											nNotificationClass						:= 11,
											aEventEnable							:= [ TRUE, TRUE, FALSE ],
											aEventMessageTextsConfig				:= [ '\/Überschritten', '\/Fehler', '\/Normal' ],
											stStartTime								:= F_BA_ToSTDateTime(DT#2010-01-01-00:00),
											bLogEnable								:= TRUE,
											aObjectPropertyReferences := [
												(iObject := AVSp, ePropertyId := PropPresentValue),
												(iObject := AVSp, ePropertyId := PropStatusFlags)]
										);
	
	
	fbNCNode							: FB_BACnet_Server_NC01 := (
											iParent									:= fbMscNode,
											sObjectName								:= '\/NC',
											sDescription							:= '\/Notification Classes'
										);
										
	EE									: FB_BACnet_EE := (
											iParent									:= fbMscNode,
											sDescription							:= '\/Event Enrollment',
											nNotificationClass						:= 11,
											aEventEnable							:= [ TRUE, TRUE, FALSE ],
											aEventMessageTextsConfig				:= [ '\/Überschritten', '\/Fehler', '\/Normal' ],
											stEventParameter						:= (
												eEventType							:= E_BACnet_EventType.eOutOfRange, 
												stEventArgs := (
													stOutOfRange := (
														nTimeDelay 					:= 0,
														fLowLimit  					:= 0.0,
														fHighLimit 					:= 200,
														fDeadband  					:= 1.0))),
											stObjectPropertyReference				:= F_BACnet_Reference(AVSp, PropPresentValue));

	(*
	NC01_Standard						: FB_BACnet_NC := (
											iParent									:= fbMscNode,
											nObjectInstance							:= 11,
											nNotificationClass						:= 11,
											sDescription							:= '\/Test NC01 Standard',
											aAckRequired							:= [ TRUE, TRUE, FALSE ],
											nPriority								:= [ 10, 11, 12 ]);
	NC02_Extended						: FB_BACnet_NC := (
											iParent									:= fbMscNode,
											nObjectInstance							:= 10,
											nNotificationClass						:= 10,
											sDescription							:= '\/Test NC02 Extended',
											aAckRequired							:= [ TRUE, TRUE, TRUE ],
											nPriority								:= [ 13, 14, 15 ]);
	*)
	
	{attribute 'hide'}
	_stUnusedCmpData					: ST_BACnet_Destination;
	nCompareRecipient_Index				: UINT										:= 0;
	NC03_RecipientTest					: FB_BACnet_NC := (
											iParent									:= fbMscNode,
											nObjectInstance							:= 244,
											nNotificationClass						:= 244,
											sDescription							:= '\/Test NC03 RecipientTest',
											aAckRequired							:= [ TRUE, TRUE, FALSE ],
											aPriority								:= [ 224, 223, 222 ],
											aRecipientList	:= 
												[
													(
														stValidDays					:= (bSunday:=TRUE, bSaturday:=TRUE, bFriday:=TRUE),
														stFromTime					:= F_BA_ToSTTime(T#0H),
														stToTime					:= F_BA_ToSTTime(T#23H59M59S),
														stRecipient					:= F_BACnet_DeviceRecipient(nDeviceInstance:=5),
														nProcessId					:= 20100,
														bIssueConfirmed				:= FALSE
													),
													(
														stValidDays					:= (bSunday:=TRUE, bSaturday:=TRUE),
														stFromTime					:= F_BA_ToSTTime(T#0H),
														stToTime					:= F_BA_ToSTTime(T#23H59M59S),
														stRecipient					:= F_BACnet_EthernetRecipient(nIPAddress1:=192,168,10,200, nPort:=47808, nNetworkNr:=444),
														nProcessId					:= 30100,
														bIssueConfirmed				:= TRUE
													)
													(* (
														stValidDays					:= (bSunday:=TRUE, bSaturday:=TRUE, bFriday:=TRUE),
														stFromTime					:= F_BA_ToSTTime(T#0H),
														stToTime					:= F_BA_ToSTTime(T#23H59M59S),
														stRecipient := (
															eRecipientChoice		:= E_BACnet_RecipientChoice.eDevice,
															aEntry := (
																tDeviceId			:= 20,
																stNetAddr := (
																	eChoice			:= E_BACnet_AddressChoice.eEthernet,
																	eAddress		:= [ 10, 10, 10, 10, 10, 10, 1, 1 ],
																	nNetworkNr		:= 0))),
														nProcessId					:= 20100,
														bIssueConfirmed				:= FALSE
													) *)
												]
											);
END_VAR
// --- Special: ---------------------------------------------------------------------------------------------------------------------------------------
VAR_INPUT		
	fbSpcNode							: FB_BACnet_View := (
											iParent									:= fbLibNode,
											eNodeType								:= E_BACnet_NodeType.eArea,
											sObjectName								:= '\/Spec',
											sDescription							:= '\/Special');
											
	Acc01								: FB_BACnet_Acc := (
											iParent									:= fbSpcNode,
											sDescription							:= '\/Accumulator');
	Acc02								: FB_BACnet_Acc_IO := (
											iParent									:= fbSpcNode,
											sDescription							:= '\/Accumulator I/O');
											
	PC01								: FB_BACnet_PC_Raw := (
											iParent									:= fbSpcNode,
											sDescription							:= '\/Pulse Converter');
											
	Prog01								: FB_BACnet_Prog := (
											iParent									:= fbSpcNode,
											sDescription							:= '\/Program');
END_VAR
// --- Primitive Value Objects: ---------------------------------------------------------------------------------------------------------------------------------------
VAR_INPUT		
	fbPrmNode							: FB_BACnet_View := (
											iParent									:= fbLibNode,
											eNodeType								:= E_BACnet_NodeType.eArea,
											sObjectName								:= '\/Primitive',
											sDescription							:= '\/Primitive');
										
	fbInt								: FB_BACnet_INT := (
											iParent									:= fbPrmNode,
											sDescription							:= '\/Signed Integer Value',
											nValue									:= -42);
	fbLav								: FB_BACnet_LAV := (
											iParent									:= fbPrmNode,
											sDescription							:= '\/Large Analog Value',
											fValue									:= 17E42);											
	fbString							: FB_BACnet_String := (
											iParent									:= fbPrmNode,
											sDescription							:= '\/String Value',
											sValue									:= 'A simple string value');											
	fbUInt								: FB_BACnet_UINT := (
											iParent									:= fbPrmNode,
											sDescription							:= '\/Unsigned Integer Value',
											nValue									:= 42 );
END_VAR
// --- Tests: ---------------------------------------------------------------------------------------------------------------------------------------
VAR_INPUT		
	fbTestNode							: FB_BACnet_View := (
											iParent									:= fbLibNode,
											eNodeType								:= E_BACnet_NodeType.eArea,
											sObjectName								:= '\/Tst',
											sDescription							:= '\/Tests');
										
	nOffsetInstID						: UDINT										:= 402;	
	ChangeInstAV1						: FB_BACnet_AV_Setp := (
											iParent									:= fbTestNode,
											nObjectInstance							:= 1+nOffsetInstID);
	ChangeInstAV2						: FB_BACnet_AV_Setp := (
											iParent									:= fbTestNode,
											nObjectInstance							:= 2+nOffsetInstID);
	ChangeInstAV3						: FB_BACnet_AV_Setp := (
											iParent									:= fbTestNode,
											nObjectInstance							:= 3+nOffsetInstID);
END_VAR

fbLibNode();
IF (fbLibNode.bUpdateCOV) THEN
	nLibNode_UpdateCount := (nLibNode_UpdateCount+1);
END_IF

// Analog:
fbANode();
AV();
AV5P(bEnSfty := AV5P_TestEnSfty);
AVDsp();
AVSp();
AI_TSenRaw(nRawState:=AI_TSenRaw_State, nRawVal:=AI_TSenRaw_DataIn);
AI_TSenProc(fVal:=AI_TSenProc_Value);
AI_TSenIO();
AIDsp_TSenIO();
AO_Cmd(eRlbtyPgm:=AO_Cmd_RlbtyPgm, bRawOvrrd:=AO_Cmd_RawOvrrd);
AO_CmdRaw(nRawVal=>AO_CmdRaw_Out);
AO_CmdIORaw();
AO_Cmd5P(eRlbtyPgm:=AO_Cmd5P_RlbtyPgm, bRawOvrrd:=AO_Cmd5P_RawOvrrd);
AO_CmdRaw5P(bRawOvrrd:=(AO_CmdRaw5P_State<>0), nRawVal=>AO_CmdRaw5P_Out);
AO_CmdIO5P();
AODisp_CmdIO5P();
AO_CmdIO();

// Binary:
fbBNode();

BV();
BV5P();
BVDsp();
BVSp();
BI_DstbRaw(bRawVal:=BI_DstbRaw_In);
BI_DstbIO();
BIDsp_SwiIO();
BO_Cmd(eRlbtyPgm:=BO_Cmd_RlbtyPgm, bRawOvrrd:=BO_Cmd_RawOvrrd);
BO_CmdRaw(bRawVal=>BO_CmdRaw_Out);
BO_CmdIO();
BO_Cmd5P(eRlbtyPgm:=BO_Cmd5P_RlbtyPgm, bRawOvrrd:=BO_Cmd5P_RawOvrrd);
BO_CmdRaw5P(bRawVal=>BO_CmdRaw5P_Out, bEnFdbck:=TRUE, bRawValFdbck:=BO_CmdRaw5P_Feedback, bRawOvrrd:=BO_CmdRaw5P_OverrIO);
BO_CmdIO5P();
BODisp_CmdIO5P();

// Multistate:
fbMNode();

MV();
MV5P();
MVDsp();
MVSp();
MI_StateRaw(nRawValue:=MI_StateRaw_In);
MI_StateIO();
MIDsp_Swi_StateRaw(nRawValue:=MIDsp_Swi_StateRaw_In);
MO_Cmd(bRawOvrrd:=MO_Cmd_RawOvrrd);
MO_CmdRaw(nRawValue=>MO_CmdRaw_Out);
MO_5P(bRawOvrrd:=MO_5P_RawOvrrd);
MO_Raw5P(nRawValue=>MO_Raw5P_Out);
MODisp_Raw5P(nRawValue=>MODisp_Raw5P_Out);
MODisp_IO5P();

// Misc:
fbMscNode();

Dev01();

File01();
LOOP();
fbLoopRefNode();
LoopRef_Setpt();
LoopRef_CtrlVar();
LoopRef_Y();
LoopRef();
CAL01();
CAL02();
CAL03();
SchedA();
IF (SchedB_AssignTestCal2Reference) THEN
	SchedB_AssignTestCal2Reference := FALSE;
	SchedB.aCalendar[2].iRefCalendar := CAL01;
	SchedB.aCalendar[2].aEntry := F_BACnet_SchedEntry1xB(T#11H, TRUE);
END_IF
SchedB();
SchedM();
EventLog_NC11();
EventLog_NC12();
IF (TLog_AssignTestReference) THEN
	TLog_AssignTestReference := FALSE;
	TLog.stObjectPropertyReference.iObject := SchedA;
	TLog.ObjectPropertyReference := TLog.stObjectPropertyReference;
END_IF
IF (TLog_ReadReference) THEN
	TLog_ReadReference := FALSE;
	_hRes := TLog.ReadPropertyReference(E_BACnetPropIdentifier.PropLogDeviceObjectProperty, TLog.stObjectPropertyReference);
	F_BA_LogMessage1(ADSLOG_MSGTYPE_ERROR, 'DEBUG73', 'Read TLog-Ref: Result=0x%x', F_DINT(_hRes));		
END_IF
IF (TLog_LogReferenceInfo) THEN
	TLog_LogReferenceInfo := FALSE;
	IF (TLog.stObjectPropertyReference.iObject = 0) THEN
		F_BA_LogMessage(ADSLOG_MSGTYPE_ERROR, 'DEBUG80', 'TLog-Ref: 0');
	ELSE
		tTemp := TLog.stObjectPropertyReference.iObject.ObjectName;
		F_BA_LogMessage1(ADSLOG_MSGTYPE_ERROR, 'DEBUG83', 'TLog-Ref: %s', F_STRING(tTemp));
	END_IF
END_IF
TLog();
TLogCov();
TLogNoRef();
TLogM();

EE();

fbNCNode();
(*
NC01_Standard();
NC02_Extended();
*)
IF (nCompareRecipient_Index <> 0) THEN
	F_BA_Print('Compare Recipient [Unused]', ADR(_stUnusedCmpData), SIZEOF(ST_BACnet_Destination), TRUE, 64);
	F_BA_Print('Compare Recipient [Index]', ADR(NC03_RecipientTest.aRecipientList[nCompareRecipient_Index]), SIZEOF(ST_BACnet_Destination), TRUE, 64);
	
	nCompareRecipient_Index := TO_UINT(F_BA_GetUsedEntryCount(ADR(NC03_RecipientTest.aRecipientList), 1, BACnet_Param.nNC_RecipientListSize, _stUnusedCmpData));
	F_BA_LogMessage1(ADSLOG_MSGTYPE_ERROR, 'Compare Recipient', 'Recipient Count: %d', F_UINT(nCompareRecipient_Index));
	
	nCompareRecipient_Index := 0;
END_IF
NC03_RecipientTest();

// Special:
fbSpcNode();

Acc01();
Acc02();
PC01();
Prog01();

// Primitive Value
fbPrmNode();
fbInt();
fbLav();
fbString();
fbUInt();

// Test:
fbTestNode();

ChangeInstAV1();
ChangeInstAV2();
ChangeInstAV3();

END_PROGRAM

// TEST/TestPackage/PERFORMANCE_MIX
PROGRAM PERFORMANCE_MIX
VAR
	i : UDINT;
	bPerf : BOOL := TRUE;
	bOriginal : BOOL := FALSE;
	aAV   : ARRAY[0..199] OF FB_BACnet_AV;
	aBV   : ARRAY[0..199] OF FB_BACnet_BV;
	aMV   : ARRAY[0..199] OF FB_BACnet_MV;
	aBI   : ARRAY[0..99] OF FB_BACnet_BI_IO;
	aAI   : ARRAY[0..49] OF FB_BACnet_AI;
	aAO  	: ARRAY[0..49] OF FB_BACnet_AO_IO;
	aBO   : ARRAY[0..49] OF FB_BACnet_BO_IO;
	aMI   : ARRAY[0..49] OF FB_BACnet_MI_IO;
	aMO   : ARRAY[0..49] OF FB_BACnet_MO_IO;
	aSCH  : ARRAY[0..19] OF FB_BACnet_SchedB;
	aTLOG : ARRAY[0..19] OF FB_BACnet_TLog;
	aCAL  : ARRAY[0..1] OF FB_BACnet_Cal;
	aNC   : ARRAY[0..4] OF FB_BACnet_NC;
END_VAR

IF bPerf THEN
	FOR i := 0 TO 199 DO
		aAV[i]( );
		aBV[i]( );
		aMV[i]( );
	END_FOR
	
	IF NOT bOriginal THEN
		FOR i := 0 TO 99 DO
			aBI[i]();
		END_FOR
		
		FOR i := 0 TO 49 DO
			aAI[i]();
			aAO[i]();
			aBO[i]();
			aMI[i]();
			aMO[i]();	
		END_FOR
		
		FOR i := 0 TO 19 DO
			aSCH[i]();
			aTLOG[i]();
		END_FOR
		
		FOR i := 0 TO 1 DO
			aCAL[i]();
		END_FOR
		
		FOR i := 0 TO 4 DO
			aNC[i]();
		END_FOR
	END_IF
END_IF

END_PROGRAM

// TEST/TestPackage/DYN_OBJECTS
// See 'FB_BACnet_DynObjectManager' for more information.
PROGRAM DYN_OBJECTS
VAR
	fbDynObject	: FB_BACnet_DynObjectManager		:= (bCycleObjects := TRUE);
	
	bCreate		: BOOL;
	bDelete		: BOOL;
	
	DynView		: POINTER TO FB_BACnet_View;
	DynAV01		: POINTER TO FB_BACnet_AV;
	DynAV02		: POINTER TO FB_BACnet_SmplAV01;
END_VAR
VAR
	nCounter	: UDINT;
END_VAR

// Management FB has to be called cyclic:
fbDynObject();

IF (fbDynObject.Ready) THEN
	IF (bCreate) THEN
		bCreate := FALSE;
		
		// [Variant 1] Create standard object types:
		IF (fbDynObject.CreateObject(DynView, E_BACnet_CreateObjType.eStructuredView, BACnet_Globals.nBACnetInstId_Auto, 'DynView', 'Dynamic View', 0)) THEN
			// [Optional] ...
		END_IF
		IF (fbDynObject.CreateObject(DynAV01, E_BACnet_CreateObjType.eAnalogValue, BACnet_Globals.nBACnetInstId_Auto, '\/DynAV01', '\/Dynamic AV 1', DynView)) THEN
			// [Optional] ...
		END_IF
		
		// [Variant 2] Create objects of derived types:
		DynAV02 := __NEW(FB_BACnet_SmplAV01);
		IF (fbDynObject.CreateObjectEx(DynAV02, BACnet_Globals.nBACnetInstId_Auto, '\/DynAV02', '\/Dynamic AV 2', DynView)) THEN
			// [Optional] ...
		END_IF
	END_IF
	
	IF (bDelete) THEN
		bDelete := FALSE;
		
		// [Variant 1] Delete all objects comfortably via object manager: 
		fbDynObject.Reset();

		// [Variant 2] Delete all objects manually:
		(*
		fbDynObject.DeleteObject(DynAV01);
		fbDynObject.DeleteObject(DynAV02);
		fbDynObject.DeleteObject(DynView);
		*)
	END_IF

	// Sample PLC code:
	// > Take care of valid object pointers!
	IF (fbDynObject.CreatedObjects > 0) THEN
		nCounter := (nCounter+1);
		
		// Simulate changing value:
		DynAV01^.bEnPgm := TRUE;
		DynAV01^.fValPgm := (TO_REAL(nCounter MOD 1000)/100);
		DynAV02^.bEnPgm := TRUE;
		DynAV02^.fValPgm := (DynAV01^.fValPgm+2.2);
		
		// [Variant 2] Call created objecty manually
		IF (NOT fbDynObject.bCycleObjects) THEN
			DynView^();
			DynAV01^();
			DynAV02^();
		END_IF
	END_IF
END_IF

END_PROGRAM

// TEST/CLIENT_Andreas
PROGRAM CLIENT_Andreas
VAR
	fbClientFb : FB_ClientTest := (Client := (nDeviceInstance := 1));	
	fbClientFb2 : FB_ClientTest := (Client := (nDeviceInstance := 1));	
	
	fbClient : FB_BACnet_Client := (nDeviceInstance := 3776986, eReadMode:=E_BACnet_CommMode.eRp);
//	fbDevice : FB_BACnetRM_DeviceVisu := (Client:=fbClient);
	fbAo : FB_BACnetRM_AO := (Client:=fbClient, nObjectInstance:=0);
	fbAv : FB_BACnetRM_AV := (Client:=fbClient, nObjectInstance:=0);
	fbBi : FB_BACnetRM_BI := (Client:=fbClient, nObjectInstance:=0);
	fbBo : FB_BACnetRM_BO := (Client:=fbClient, nObjectInstance:=11001);
	
//	fbVisAv0 : FB_BACnetRM_VisuAV := (Client:=fbClient, nObjectInstance:=0);
//	fbVisAv1 : FB_BACnetRM_VisuAV := (Client:=fbClient, nObjectInstance:=1);
//	fbVisAv2 : FB_BACnetRM_VisuAV := (Client:=fbClient, nObjectInstance:=2);
//	fbVisAv3 : FB_BACnetRM_VisuAV := (Client:=fbClient, nObjectInstance:=3);
	
	diag : ST_BACnet_Diagnosis;
	scanRes : ARRAY [0..99] OF ST_BACnetRM_ScanResult;
	syncTime : ST_BA_DateTime;
	
	bDiag : BOOL;
	bScan : BOOL;
	bGet : BOOL;
	bSync : BOOL;
	
	fbClient2 : FB_BACnet_Client := (nDeviceInstance := 546);
	
	c : FB_BACnet_Client := (nDeviceInstance:=163719);
	sObjectName : STRING;
	fbRead  : FB_BACnetRM_ReadPropertyEx  := (Client:=c, pData:=ADR(sObjectName), nData:=255, ePropID:=PropObjectName, eObjType:=ObjMultiStateValue, nObjInst:=10000);
	fbWrite : FB_BACnetRM_WritePropertyEx := (Client:=c, pData:=ADR(sObjectName), nData:=255, ePropID:=PropObjectName, eObjType:=ObjMultiStateValue, nObjInst:=10000);
END_VAR

fbClientFb();
fbClientFb2();
fbClient();
//fbDevice();
fbAv();
FbAo();
fbBi();
fbBo();
//fbVisAv0();
//fbVisAv1();
//fbVisAv2();
//fbVisAv3();

fbClient2();

IF bDiag THEN
	fbClient.Adapter.GetDiagnosis(ADR(diag));
END_IF

IF bScan THEN	
	fbClient.Adapter.StartScan();
	bScan:=FALSE;
END_IF

IF bGet THEN
	fbClient.Adapter.GetScanResult(ADR(scanRes), 100);
	bGet:=FALSE;
END_IF

IF bSync THEN
	fbClient.Adapter.TimeSync(ADR(syncTime), TRUE);
	bSync:=FALSE;
END_IF

fbRead();
fbWrite();
c();

END_PROGRAM

// TEST/CLIENT_Marco
PROGRAM CLIENT_Marco
VAR
	fbClient			: FB_BACnet_Client					:= (nDeviceInstance := 3776986(*, eReadMode := E_BACnet_CommMode.eCov*));
	
//	AV01				: FB_BACnetRM_ExpAV01				:= (Client := fbClient, nObjectInstance := 12011);
//	AV02				: FB_BACnetRM_ExpAV02				:= (Client := fbClient, nObjectInstance := 12011);
	AV03				: FB_BACnetRM_SmplAV01				:= (Client := fbClient, nObjectInstance := 12011);
//	SchedM				: FB_BACnetRM_SchedM				:= (Client := fbClient, nObjectInstance := 12101);
END_VAR

fbClient();

//AV01();
//AV02();
AV03();
//SchedM();

END_PROGRAM

// TEST/Experimental
PROGRAM Experimental
VAR
	fbExpNode							: FB_BACnet_View := (
											sObjectName								:= '\/ExpNode',
											sDescription							:= '\/Test Experimental Node');
END_VAR
VAR
//	TLogMulti							: FB_BACnet_ExpTLM := (
//											iParent									:= fbExpNode,
//											sDescription							:= '\/Trend Multiple',
//											nNotificationClass						:= 11);

	TLog_AVSp							: FB_BACnet_AV_Setp := (
											iParent									:= fbExpNode,
											sDescription							:= '\/Trendlog AV Setpoint',
											eUnit									:= E_BA_Unit.eTime_Hours,
											fValue									:= 168);
	TLog								: FB_BACnet_ExpTLog := (
											iParent									:= fbExpNode,
											sDescription							:= '\/Trendlog',
											stObjectPropertyReference				:= F_BACnet_Reference(TLog_AVSp, PropPresentValue),
											nNotificationClass						:= 11);
END_VAR

fbExpNode();

//TLogMulti();

TLog_AVSp();
TLog();

END_PROGRAM

// TEST/MAIN
PROGRAM MAIN

// Test Programs:
//CLIENT_Andreas();

//Experimental();

//FB_MAIN();
//PRG_MAIN();
//TEMP();

// TestPackage:
//_MAIN();

//fbNC();
RT();

END_PROGRAM

// TEST/TEMP
PROGRAM TEMP
VAR
	View					: FB_BACnet_View := (
								sDescription							:= '\/View');
	MyAV1					: FB_BACnet_AV := (
								iParent									:= View,
								sDescription							:= '\/My AV 1');
	MyAV2					: FB_BACnet_AV := (
								iParent									:= View,
								sDescription							:= '\/My AV 1');
			                
	SubView					: FB_BACnet_View := (
								iParent									:= View,
								sDescription							:= '\/Sub View');
	MySubAV1				: FB_BACnet_AV := (
								iParent									:= SubView,
								sDescription							:= '\/My Sub AV 1');
	MySubAV2				: FB_BACnet_AV := (
								iParent									:= SubView,
								sDescription							:= '\/My Sub AV 1');								
END_VAR

View();
MyAV1();
MyAV2();

SubView();
MySubAV1();
MySubAV2();

END_PROGRAM
